(* CoDeSys 2.3.9.62 project: PuertaGaraje.pro *)
(* Libraries: Standard.lib 2.6.14 10:37:46 *)

(* Global variable list: Global_Variables *)
VAR_GLOBAL

   (* Entradas *)
   P : BOOL;
   FCA:BOOL;
  FCC: BOOL;

   (* Salidas *)
   Abrir: BOOL;
   Cerrar : BOOL;

END_VAR

(* POU PLC_PRG, ST *)
PROGRAM PLC_PRG
VAR
END_VAR
Animacion();
ControlLD();
END_PROGRAM

(* POU Animacion, ST *)
PROGRAM Animacion
VAR
    Pos : INT;
END_VAR
IF (Abrir AND Pos>-160) THEN
   Pos:=Pos-3;
END_IF

IF (Cerrar AND POS<0) THEN
   Pos:=Pos+3;
END_IF

FCC:= (Pos>=0) ;
FCA:=(Pos<=-160);
END_PROGRAM

(* POU ControlLD, LD *)
PROGRAM ControlLD
VAR
	E0:BOOL;
	E1:BOOL;
	E2:BOOL;
	E3:BOOL;
	E4:BOOL;
	E5:BOOL;
	E6:BOOL;
END_VAR
VAR (* helpers for the ST form of the networks *)
	_p1 : BOOL;
	_p2 : BOOL;
	_p3 : BOOL;
	_p4 : BOOL;
	_p5 : BOOL;
	_p6 : BOOL;
	_p7 : BOOL;
	_p8 : BOOL;
	_p9 : BOOL;
END_VAR
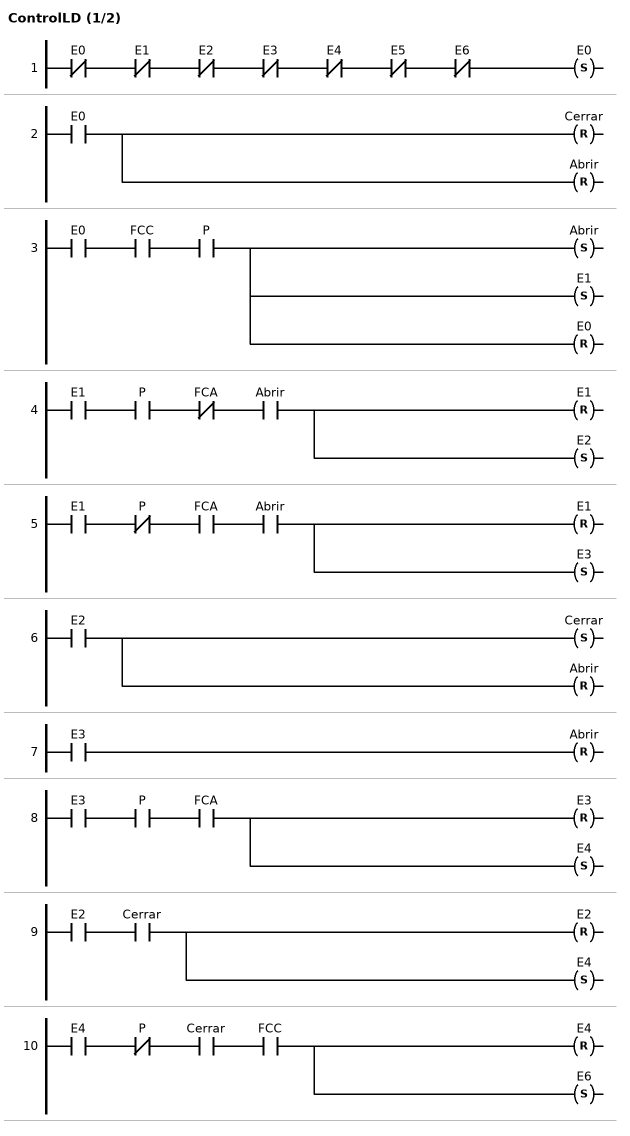
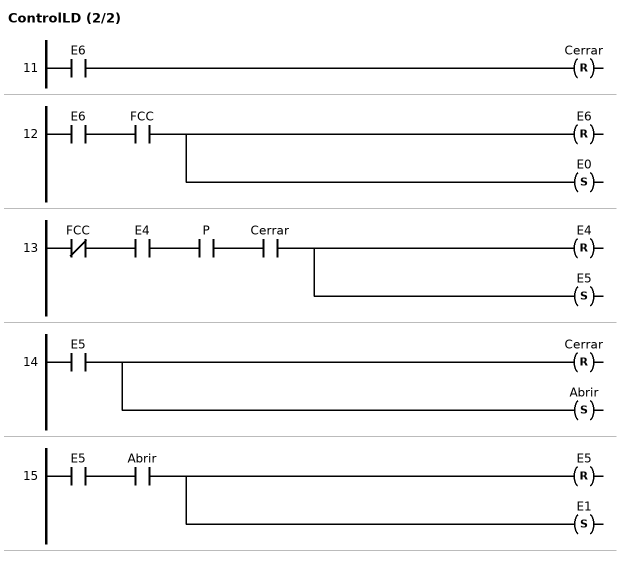
_LD_ (* Ladder Diagram *)
NETWORK 1
	[/E0] - [/E1] - [/E2] - [/E3] - [/E4] - [/E5] - [/E6] --- (S E0)
NETWORK 2
	[E0] --- (R Cerrar) (R Abrir)
NETWORK 3
	[E0] - [FCC] - [P] --- (S Abrir) (S E1) (R E0)
NETWORK 4
	[E1] - [P] - [/FCA] - [Abrir] --- (R E1) (S E2)
NETWORK 5
	[E1] - [/P] - [FCA] - [Abrir] --- (R E1) (S E3)
NETWORK 6
	[E2] --- (S Cerrar) (R Abrir)
NETWORK 7
	[E3] --- (R Abrir)
NETWORK 8
	[E3] - [P] - [FCA] --- (R E3) (S E4)
NETWORK 9
	[E2] - [Cerrar] --- (R E2) (S E4)
NETWORK 10
	[E4] - [/P] - [Cerrar] - [FCC] --- (R E4) (S E6)
NETWORK 11
	[E6] --- (R Cerrar)
NETWORK 12
	[E6] - [FCC] --- (R E6) (S E0)
NETWORK 13
	[/FCC] - [E4] - [P] - [Cerrar] --- (R E4) (S E5)
NETWORK 14
	[E5] --- (R Cerrar) (S Abrir)
NETWORK 15
	[E5] - [Abrir] --- (R E5) (S E1)
_END_LD_
(* the same logic as Structured Text *)
(* Network 1 *)
IF NOT E0 AND NOT E1 AND NOT E2 AND NOT E3 AND NOT E4 AND NOT E5 AND NOT E6 THEN E0 := TRUE; END_IF;
(* Network 2 *)
IF E0 THEN Cerrar := FALSE; Abrir := FALSE; END_IF;
(* Network 3 *)
_p1 := E0 AND FCC AND P;
IF _p1 THEN Abrir := TRUE; E1 := TRUE; E0 := FALSE; END_IF;
(* Network 4 *)
_p2 := E1 AND P AND NOT FCA AND Abrir;
IF _p2 THEN E1 := FALSE; E2 := TRUE; END_IF;
(* Network 5 *)
_p3 := E1 AND NOT P AND FCA AND Abrir;
IF _p3 THEN E1 := FALSE; E3 := TRUE; END_IF;
(* Network 6 *)
IF E2 THEN Cerrar := TRUE; Abrir := FALSE; END_IF;
(* Network 7 *)
IF E3 THEN Abrir := FALSE; END_IF;
(* Network 8 *)
_p4 := E3 AND P AND FCA;
IF _p4 THEN E3 := FALSE; E4 := TRUE; END_IF;
(* Network 9 *)
_p5 := E2 AND Cerrar;
IF _p5 THEN E2 := FALSE; E4 := TRUE; END_IF;
(* Network 10 *)
_p6 := E4 AND NOT P AND Cerrar AND FCC;
IF _p6 THEN E4 := FALSE; E6 := TRUE; END_IF;
(* Network 11 *)
IF E6 THEN Cerrar := FALSE; END_IF;
(* Network 12 *)
_p7 := E6 AND FCC;
IF _p7 THEN E6 := FALSE; E0 := TRUE; END_IF;
(* Network 13 *)
_p8 := NOT FCC AND E4 AND P AND Cerrar;
IF _p8 THEN E4 := FALSE; E5 := TRUE; END_IF;
(* Network 14 *)
IF E5 THEN Cerrar := FALSE; Abrir := TRUE; END_IF;
(* Network 15 *)
_p9 := E5 AND Abrir;
IF _p9 THEN E5 := FALSE; E1 := TRUE; END_IF;
END_PROGRAM

(* Visualisation Visu
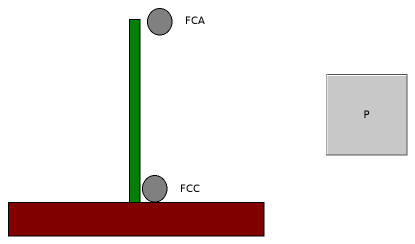
button at (450,140)-(531,221): text "P"; taps P
rectangle at (253,85)-(264,269): bottom Animacion.Pos
ellipse at (266,241)-(291,268): alarm colour if FCC
ellipse at (271,74)-(296,101): alarm colour if FCA
rectangle at (286,244)-(342,265): text "FCC"
rectangle at (291,76)-(347,97): text "FCA"
1 more shapes without text or variables
*)
